// TIA Portal project "SCL DESESCALADO" (V11)

(* hardware
DEVICE "S7300/ET200 station_1"  SIMATIC 300-Station
   slot 0: "Perfil soporte_0"  Rail  6ES7 390-1***0-0AA0
   slot 2: "PLC_1"  CPU 313C-2 DP  6ES7 313-6CF03-0AB0  V2.6
      slot 0: "Interfaz MPI_1"  MPI
      slot 1: "Interfaz DP_1"  DP
      slot 2: "DI16/DO16_1"  DI16/DO16
      slot 4: "Contaje_1"  Counter
*)

// ===== PLC "PLC_1"  CPU 313C-2 DP =====

VAR_GLOBAL   // PLC tag table "Tabla de variables estándar"
   "Tag_1" AT %E0.0 : Bool;
   "Tag_2" AT %MD0 : Real;
   "Tag_3" AT %MD4 : Real;
END_VAR

DATA_BLOCK "DESESCALADO_DB"   // DB1
{ S7_Optimized_Access := 'FALSE' }
VERSION : 0.1
// stored: InstanceOfName DESESCALADO
"DESESCALADO"
BEGIN
END_DATA_BLOCK

FUNCTION_BLOCK "DESESCALADO"   // FB1, SCL
{ S7_Optimized_Access := 'FALSE' }
VERSION : 0.1
   VAR_INPUT
      Y2 : Real;
      Y1 : Real;
      X2 : Real;
      X1 : Real;
      calcular : Bool;
      YSEÑALANALOGICA : Real;
      "XSEÑAL ANAOLOGICA" : Real;
   END_VAR
   VAR_OUTPUT
      YESCALADO : Real;
      XDESESCALADO : Real;
   END_VAR
   VAR
      "PENDIENTE (m)" : Real;
      "PUNTOCORTE (n)" : Real;
      Y : Real;
   END_VAR
BEGIN
   IF #calcular THEN
     #"PENDIENTE (m)":= ( #Y2 - #Y1) / ( #X2 - #X1);
     #"PUNTOCORTE (n)"  := #Y2 - (#"PENDIENTE (m)" * #X2) ;
     #YESCALADO :=( #"PENDIENTE (m)" * #"XSEÑAL ANAOLOGICA") + #"PUNTOCORTE (n)";
   END_IF;

   IF #calcular  THEN
    #"PENDIENTE (m)":= ( #Y2 - #Y1) / ( #X2 - #X1);
     #"PUNTOCORTE (n)"  := #Y2 - (#"PENDIENTE (m)" * #X2) ;
     #XDESESCALADO:= ( #YSEÑALANALOGICA - #"PUNTOCORTE (n)") / #"PENDIENTE (m)" ;
     END_IF;
END_FUNCTION_BLOCK

ORGANIZATION_BLOCK "Main"   // OB1, LAD
TITLE = "Main Program Sweep (Cycle)"
{ S7_Optimized_Access := 'FALSE' }
VERSION : 0.1
   VAR_TEMP
      OB1_EV_CLASS : Byte;   // Bits 0-3 = 1 (Coming event), Bits 4-7 = 1 (Event class 1)
      OB1_SCAN_1 : Byte;   // 1 (Cold restart scan 1 of OB 1), 3 (Scan 2-n of OB 1)
      OB1_PRIORITY : Byte;   // Priority of OB Execution
      OB1_OB_NUMBR : Byte;   // 1 (Organization block 1, OB1)
      OB1_RESERVED_1 : Byte;   // Reserved for system
      OB1_RESERVED_2 : Byte;   // Reserved for system
      OB1_PREV_CYCLE : Int;   // Cycle time of previous OB1 scan (milliseconds)
      OB1_MIN_CYCLE : Int;   // Minimum cycle time of OB1 (milliseconds)
      OB1_MAX_CYCLE : Int;   // Maximum cycle time of OB1 (milliseconds)
      OB1_DATE_TIME : Date_And_Time;   // Date and time OB1 started
   END_VAR
BEGIN

REGION Network 1
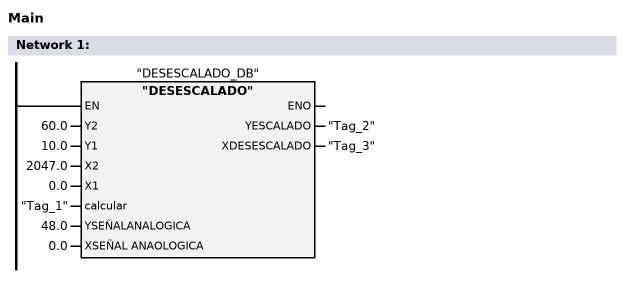
   RUNG wire#powerrail
      "DESESCALADO_DB"(Y2 := 60.0, Y1 := 10.0, X2 := 2047.0, X1 := 0.0, calcular := "Tag_1", YSEÑALANALOGICA := 48.0, "XSEÑAL ANAOLOGICA" := 0.0, YESCALADO => "Tag_2", XDESESCALADO => "Tag_3")
   END_RUNG
   // the same network as SCL:
   "DESESCALADO_DB"(Y2 := 60.0,   // "DESESCALADO"
                    Y1 := 10.0,
                    X2 := 2047.0,
                    X1 := 0.0,
                    calcular := "Tag_1",
                    YSEÑALANALOGICA := 48.0,
                    "XSEÑAL ANAOLOGICA" := 0.0,
                    YESCALADO => "Tag_2",
                    XDESESCALADO => "Tag_3");
END_REGION
END_ORGANIZATION_BLOCK